{attribute 'linkalways'} 
{attribute 'no_explicit_call' := 'This FB is a CLASS and must be accessed using methods or properties'}
{attribute 'enable_dynamic_creation'}
FUNCTION_BLOCK _ETcVnCalibrationPattern EXTENDS EnumDatatypeBase
VAR
	localData : ETcVnCalibrationPattern;
	activeData : REFERENCE TO ETcVnCalibrationPattern;
	enumBaseDatatype : _DINT(localData);
END_VAR

METHOD PRIVATE AddLocalEnumeration
VAR_INPUT
	Enumeration : T_MAXSTRING;
	Value : ETcVnCalibrationPattern;
END_VAR
AddEnumeration(Enumeration, Value);
END_METHOD

PROPERTY PUBLIC Address : PVOID
GET
Address := ADR(activeData);
END_GET
END_PROPERTY

METHOD PUBLIC ClearReference
VAR_INPUT
END_VAR
activeData REF= localData;
SetBaseDatatypeReference();
END_METHOD

METHOD PUBLIC Clone : I_Datatype
VAR
    pClone : POINTER TO _ETcVnCalibrationPattern;
END_VAR
pClone := __NEW(_ETcVnCalibrationPattern(InitialValue := Value));
Clone := pClone^;
END_METHOD

METHOD FB_init : BOOL
VAR_INPUT
	bInitRetains : BOOL; // if TRUE, the retain variables are initialized (warm start / cold start)
	bInCopyCode : BOOL;  // if TRUE, the instance afterwards gets moved into the copy code (online change)
	InitialValue : ETcVnCalibrationPattern;
END_VAR
localData := InitialValue;
AddBaseDatatype(enumBaseDatatype);
ClearReference();

AddLocalEnumeration('TCVN_CP_CIRCLES_SYM', ETcVnCalibrationPattern.TCVN_CP_CIRCLES_SYM);
AddLocalEnumeration('TCVN_CP_CIRCLES_ASYM', ETcVnCalibrationPattern.TCVN_CP_CIRCLES_ASYM);
AddLocalEnumeration('TCVN_CP_CIRCLES_ASYM_INDENT', ETcVnCalibrationPattern.TCVN_CP_CIRCLES_ASYM_INDENT);
END_METHOD

PROPERTY PUBLIC Identifier : T_MAXSTRING
GET
Identifier := 'ETcVnCalibrationPattern';
END_GET
END_PROPERTY

METHOD IsEnumeratorValueEqual : BOOL
VAR_INPUT
	Enumerator : I_KeyValueForwardEnumerator;
END_VAR
VAR
	storedValue : ETcVnCalibrationPattern;
END_VAR
IF NOT Enumerator.TryGet(storedValue) THEN
	RETURN;
END_IF

IsEnumeratorValueEqual := storedValue = activeData;
END_METHOD

METHOD PUBLIC MakeReferenceTo
VAR_INPUT
	ReferenceTarget : REFERENCE TO ETcVnCalibrationPattern;
END_VAR
activeData REF= ReferenceTarget;
SetBaseDatatypeReference();
END_METHOD

METHOD PROTECTED SetBaseDatatypeReference
VAR_INPUT
END_VAR
enumBaseDatatype.MakeReferenceTo(activeData);
END_METHOD

PROPERTY PUBLIC Size : UDINT
GET
Size := SIZEOF(activeData);
END_GET
END_PROPERTY

METHOD TryMakeReferenceTo : BOOL
VAR_INPUT
	Target : I_Datatype;
END_VAR
VAR
	targetAsEnum : I_EnumDatatype;
	pTargetData : POINTER TO ETcVnCalibrationPattern;
END_VAR
IF NOT Target.TryResolveAsEnumDatatype(targetAsEnum) THEN
	RETURN;
END_IF

IF targetAsEnum.Identifier <> Identifier THEN
	RETURN;
END_IF

pTargetData := Target.Address;
activeData REF= pTargetData^;
SetBaseDatatypeReference();
TryMakeReferenceTo := TRUE;
END_METHOD

PROPERTY PUBLIC Value : ETcVnCalibrationPattern
GET
Value := activeData;
END_GET
SET
activeData := Value;
END_SET
END_PROPERTY

END_FUNCTION_BLOCK

(* stored: Version 1.1.0.1, ProductVersion 3.1.4024.12
   POU _ETcVnCalibrationPattern: Id {be204a56-6802-0742-1c8a-00b75b63073a}, SpecialFunc None
   Folder Constructor: Id {9f20cba0-5f7a-093a-31b4-3c5b231a31b8}
   Folder Private: Id {0cd3a4ea-5fc9-0705-0107-779d99c2a4b5}
   Folder Protected: Id {5357cc1d-59d0-0e26-03ed-f2d25eea6b52}
   Method AddLocalEnumeration: Id {bd737c1b-ec38-0fa8-1a80-a9325da2d85c}
   Property Address: Id {0333ff20-2e4e-0a42-07cb-0a24edaa3db6}
   Get Get: Id {b20248e2-1a15-0097-23dd-d8cec17bed02}
   Method ClearReference: Id {0deae1ea-13a5-0fc7-30ec-b365f1a2d828}
   Method Clone: Id {2a615a63-f41d-0b41-2baa-fd52698b6ec1}
   Method FB_init: Id {dbd598fd-5bca-03ed-39d5-4be83e3130a4}
   Property Identifier: Id {5567db45-f8f4-05e5-0b26-422db8a34f4c}
   Get Get: Id {4c3c8ca8-1c0d-0d19-3ae3-2745b1e09fff}
   Method IsEnumeratorValueEqual: Id {accfae7d-c465-022d-33c5-35dfd55a6164}
   Method MakeReferenceTo: Id {6f0c2572-f70c-09de-15ad-688955501baf}
   Method SetBaseDatatypeReference: Id {f98b59c4-0303-0ac7-0fec-4d754ff90c67}
   Property Size: Id {d5efd5db-98e0-079a-3299-390ac04104de}
   Get Get: Id {c56ba355-9ebe-0d70-3e2b-0afcf55c8ff2}
   Method TryMakeReferenceTo: Id {15f1302d-7710-0073-1a8a-7a57ea134d91}
   Property Value: Id {08496045-20cb-0b60-3efd-5382a9e4e18c}
   Get Get: Id {27eece23-10c6-06fd-3e9c-298066334541}
   Set Set: Id {6daea195-8201-0af7-05c4-377c86ed0374} *)
